// Gripper without feedback sensors
FUNCTION_BLOCK FB_Gripper 
VAR_INPUT
END_VAR
VAR_OUTPUT
	bClose: BOOL;      // Output to close the grippes
END_VAR
VAR
END_VAR

// Close the gripper
METHOD Close : BOOL
VAR_INPUT
END_VAR
bClose := true; // Set output to close the gripper
END_METHOD

// Open the gripper
METHOD Open : BOOL
VAR_INPUT
END_VAR
bClose := false;  // Reset output to close the gripper
END_METHOD

END_FUNCTION_BLOCK

(* stored: Version 1.1.0.1, ProductVersion 3.1.4024.12
   POU FB_Gripper: Id {29462702-79bb-43c0-a206-6245c5a19425}, SpecialFunc None
   Method Close: Id {0f18a4f7-3c67-4762-9921-7c9c5c7e7ee4}
   Method Open: Id {cf724d07-4268-4eaa-add1-69605a6f40d4} *)
